FUNCTION Convert_UINT_TO_INT : Hresult
VAR_INPUT
	in : UINT;
	out : REFERENCE TO INT;
END_VAR
VAR
	converted : INT;
END_VAR

converted := UINT_TO_INT(in);

IF (INT_TO_UINT(converted) <> in) THEN
	Convert_UINT_TO_INT := INCOMPATIBLE;
	RETURN;
END_IF

out := converted;

END_FUNCTION

(* stored: Version 1.1.0.1, ProductVersion 3.1.4024.12
   POU Convert_UINT_TO_INT: Id {3ceea7af-f000-48b7-85c3-b59fc5c11c05}, SpecialFunc None *)
